(* PLC project  *)

FUNCTION TestCDATA

            
              x := 1;
              IF y > 0 THEN
                z := x + y;
              END_IF;
            
          
END_FUNCTION
